# EPICS substitutions: Examples/runtime.substitutions
file "db/EXAMPLE.db" {
    pattern { SYSTEM, DEVICE, PORT }
            { Beamline0, Picometer, L0 }
            { Beamline1, Picometer, L1 }
            { Beamline2, Picometer, L2 }
}
